TEXTLIST TextList_State2
  0 = 'Wait for Door Open..'
  10 = 'Wait For Part 1 Load and Cycle Start...'
  20 = 'Door Closing...'
  30 = 'Clamp CC1 CC3 CC5 Closing...'
  40 = 'Trunmion is Moving 0 to 50 Degree for Load 2'
  50 = 'Door Opening...'
  60 = 'Wait For Part 2 Load and Cycle Start...'
  70 = 'Clamp CC2 CC4 CC6 Closing..'
  80 = 'Door Closing...'
  90 = 'Trunmion is Moving 50 to 0 Degree...'
  100 = 'Turn Table Moving 0 to 180 Degree for weld Position...'
  110 = 'Robot Start....Waiting for Weld Complete 1....'
  120 = 'Trunmion is Moving 0 to 50 Degree for Weld 2...'
  130 = 'Robot Start....Waiting for Weld Complete 2....'
  140 = 'Clamp CC1 CC3 CC5 Opening...'
  150 = 'Robot Clear To Pick....Waiting for Pick Complete 1....'
  160 = 'Trunmion is Moving 0 Degree for Pick 2...'
  170 = 'Clamp CC2 CC4 CC6 Opening...'
  180 = 'Robot Clear To Pick....Waiting for Pick Complete 2....'
   = ''
END_TEXTLIST

(* stored: Version 1.1.0.1, ProductVersion 3.1.4024.16
   TextList TextList_State2: Id {de3cbfd6-428a-4c1f-b6f0-481d00e8f87a} *)
